// TIA Portal V20 export
DATA_BLOCK "CallEquipment_DB"   // DB130
{ DB_Accessible_From_OPC_UA := 'FALSE' }
// stored: AssignedProDiagFB Unit1.Em13.ProDiag, DBAccessibleFromOPCUA false, DBAccessibleFromWebserver false, InstanceOfName Unit1.Em13.CallEquipment, InstanceOfType FB, Namespace Unit1.Em13
"Unit1.Em13.CallEquipment"
   // VAR_INPUT
   //    ZoneOperationEnable { ExternalWritable := 'False'} : "LWONIK_typeSafetyZoneManualOperation";
   //    FATMode { ExternalWritable := 'False'} : "LER_TypeFATMode_ModeSelect";
   // END_VAR
   // VAR_IN_OUT
   //    unitStatus : "LAF_typeUnitStatus";
   //    emFeedback : "LUC_typeEmFeedback";
   //    unitAlarmDB : "LAF_typeAlarms";
   // END_VAR
   // VAR
   //    InstSequenceJRUnloading { ExternalWritable := 'False'} : "Unit1.Em13.Sequence_1_JRUnloading";
   //    instJRUnloadingHomeJob1 { ExternalWritable := 'False'} : "LAF_SelectJob";
   //    instJRUnloadingLoadJob2 { ExternalWritable := 'False'} : "LAF_SelectJob";
   //    instJRUnloadingCoveyorUnloadJob3 { ExternalWritable := 'False'} : "LAF_SelectJob";
   //    instJRUnloadingStackNgBoxUnloadJob4 { ExternalWritable := 'False'} : "LAF_SelectJob";
   //    instCmJRUnloadingPnPJRDetect { ExternalWritable := 'False'} : "LBC_DigitalSignalCn";
   //    instCmJRUnloadingPnPSafetyPin { ExternalWritable := 'False'} : "LBC_DigitalSignalCn";
   //    instCmJRUnloadingPnPAxisX { ExternalWritable := 'False'} : "LBC_Axis64Pos_TecPlcCn";
   //    instCmJRUnloadingPnPAxisZ { ExternalWritable := 'False'} : "LBC_Axis64Pos_TecPlcCn";
   //    instCmJRUnloadingPnPAxisC { ExternalWritable := 'False'} : "LBC_Axis64Pos_TecPlcCn";
   //    instCmJRUnloadingPnPClampOpenClose { ExternalWritable := 'False'} : "LBC_TwoWayActuatorCn";
   //    instInterlockJRUnloadingPnPAxisX { ExternalWritable := 'False'} : "LER_Axis64Pos_InterlockSummary";
   //    instInterlockJRUnloadingPnPAxisZ { ExternalWritable := 'False'} : "LER_Axis64Pos_InterlockSummary";
   //    instInterlockJRUnloadingPnPAxisC { ExternalWritable := 'False'} : "LER_Axis64Pos_InterlockSummary";
   //    instLDrv701ControlJRUnloadingPnPAxisZ { ExternalWritable := 'False'} : "LDrvSafe_SinaTlg701Control";
   //    instLDrv701StatusJRUnloadingPnPAxisZ { ExternalWritable := 'False'} : "LDrvSafe_SinaTlg701Status";
   //    instManageAlarms { ExternalWritable := 'False'} : "LAF_ManageAlarms";
   //    instEventsPFE { ExternalWritable := 'False'} : "Unit1.Em13.EventsPFE";
   //    statUnitStatus { ExternalWritable := 'False'} : "LAF_typeUnitStatus";
   //    statSlmStatus { ExternalWritable := 'False'} : Struct
   //       running : Bool;
   //       powerOff : Bool;
   //    END_STRUCT;
   //    statAllBrakeTest { ExternalWritable := 'False'} : "LER_typeBrakeTestUnitCommands";
   //    statPartData { ExternalWritable := 'False'} : "LER_typePartData";
   //    statRoutingOk { ExternalWritable := 'False'} : Array[0..99] of Bool;
   //    statRoutingNok { ExternalWritable := 'False'} : Array[0..99] of Bool;
   //    statTonTime { ExternalWritable := 'False'} : Array[0..999] of TON_TIME;
   //    statTofTime { ExternalWritable := 'False'} : Array[0..9] of TOF_TIME;
   //    statPulse { ExternalWritable := 'False'} : Array[0..999] of Bool;
   //    statEnableManualCmds { ExternalWritable := 'False'} : Bool;
   //    "*** Interlock Axis ***" : Bool;
   //    JRUnloadingPnPAxisX_Jog { S7_SetPoint := 'True'} : Array[0..2] of "LER_Axis_Jog";
   //    JRUnloadingPnPAxisZ_Jog { S7_SetPoint := 'True'} : Array[0..2] of "LER_Axis_Jog";
   //    JRUnloadingPnPAxisC_Jog { S7_SetPoint := 'True'} : Array[0..2] of "LER_Axis_Jog";
   //    JRUnloadingPnPAxisX_interlock { S7_SetPoint := 'True'} : Array[0..10] of "LER_Axis_Absolute";
   //    JRUnloadingPnPAxisZ_interlock { S7_SetPoint := 'True'} : Array[0..10] of "LER_Axis_Absolute";
   //    JRUnloadingPnPAxisC_interlock { S7_SetPoint := 'True'} : Array[0..10] of "LER_Axis_Absolute";
   //    JRUnloadingPnPAxisX_IntPos : Array[0..9] of Struct
   //       "Int" : Array[1..10] of Bool;
   //    END_STRUCT;
   //    JRUnloadingPnPAxisZ_IntPos : Array[0..9] of Struct
   //       "Int" : Array[1..10] of Bool;
   //    END_STRUCT;
   //    JRUnloadingPnPAxisC_IntPos : Array[0..9] of Struct
   //       "Int" : Array[1..10] of Bool;
   //    END_STRUCT;
   //    JRUnloadingPnPAxisX_IntHome : Array[0..9] of Bool;
   //    JRUnloadingPnPAxisZ_IntHome : Array[0..9] of Bool;
   //    JRUnloadingPnPAxisC_IntHome : Array[0..9] of Bool;
   //    JRUnloadingPnPAxisX_PosAbsolute : Array[0..10] of Bool;
   //    JRUnloadingPnPAxisZ_PosAbsolute : Array[0..10] of Bool;
   //    JRUnloadingPnPAxisC_PosAbsolute : Array[0..10] of Bool;
   //    JRUnloadingPnPAxisX_Home { S7_SetPoint := 'True'} : "LER_Axis_Homing";
   //    JRUnloadingPnPAxisZ_Home { S7_SetPoint := 'True'} : "LER_Axis_Homing";
   //    JRUnloadingPnPAxisC_Home { S7_SetPoint := 'True'} : "LER_Axis_Homing";
   //    "*** Interlock TwoWay ***" { S7_SetPoint := 'True'} : "LER_Axis_Homing";
   //    instCmJRUnloadingPnPClampOpenCloseInterlock { S7_SetPoint := 'True'} : Array[0..2] of "LER_Actuator";
   //    JRUnloadingPnPClampOpenClose_Inpos : Array[0..2] of Struct
   //       "Int" : Array[1..10] of Bool;
   //    END_STRUCT;
   //    citi_Ptrig : Array[0..20] of Bool;
   //    citiTon : Array[0..20] of TON_TIME;
   //    citi : Time;
   //    citiTest : Array[0..20] of Bool;
   // END_VAR
BEGIN
END_DATA_BLOCK
